SUBAPPLICATION Uebung_028 (* Analog-Eingang *)
  (* Standard: 61499-2 *)
  (* Version 1.0, 2023-10-23, franz *)
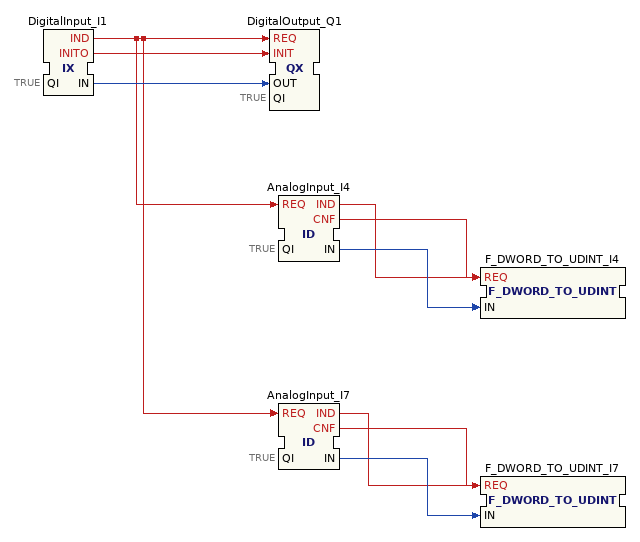
  FBS
    DigitalOutput_Q1 : QX(QI := TRUE);
    DigitalInput_I1 : IX(QI := TRUE);
    AnalogInput_I4 : ID(QI := TRUE);
    AnalogInput_I7 : ID(QI := TRUE);
    F_DWORD_TO_UDINT_I7 : F_DWORD_TO_UDINT;
    F_DWORD_TO_UDINT_I4 : F_DWORD_TO_UDINT;
  END_FBS
  EVENT_CONNECTIONS
    DigitalInput_I1.IND TO DigitalOutput_Q1.REQ;
    DigitalInput_I1.INITO TO DigitalOutput_Q1.INIT;
    AnalogInput_I7.IND TO F_DWORD_TO_UDINT_I7.REQ;
    AnalogInput_I4.IND TO F_DWORD_TO_UDINT_I4.REQ;
    DigitalInput_I1.IND TO AnalogInput_I4.REQ;
    DigitalInput_I1.IND TO AnalogInput_I7.REQ;
    AnalogInput_I7.CNF TO F_DWORD_TO_UDINT_I7.REQ;
    AnalogInput_I4.CNF TO F_DWORD_TO_UDINT_I4.REQ;
  END_CONNECTIONS
  DATA_CONNECTIONS
    DigitalInput_I1.IN TO DigitalOutput_Q1.OUT;
    AnalogInput_I7.IN TO F_DWORD_TO_UDINT_I7.IN;
    AnalogInput_I4.IN TO F_DWORD_TO_UDINT_I4.IN;
  END_CONNECTIONS
END_SUBAPPLICATION
